{attribute 'qualified_only'}
VAR_GLOBAL
END_VAR

(* stored: Version 1.1.0.1, ProductVersion 3.1.4024.16
   GVL Test: Id {0addc07b-3084-48cc-baed-d473b86d10ee} *)
